// TwinCAT 3 PLC project PLC_ElevatorControl
// ProgramVersion: 3.1.4024.12
// libraries:
//   Tc2_Standard, * (Beckhoff Automation GmbH)
//   Tc2_System, * (Beckhoff Automation GmbH)
//   Tc3_Module, * (Beckhoff Automation GmbH)
//   VisuSymbols,3.5.10.0,System
// project tree:
//   DUTs/ ElevatorOpMode.TcDUT, LiftMovingDirection.TcDUT, txt_opMode.TcTLO
//   / GlobalTextList.TcGTLO, PlcTask.TcTTO, Visualisierungsmanager.TcVMO (not stored)
//   GVLs/ GVL_LiftProj.TcGVL
//   POUs/ FB_ElevatorCtrl.TcPOU, MAIN.TcPOU
//   POUs/POU_ActuatorCtrl/ FB_DriveSimpleDoor.TcPOU, FB_DriveWinch.TcPOU, IF_DriveConstVel.TcIO, IF_DriveVariableVel.TcIO
//   POUs/POU_SequenceCtrl/ FB_move2Level.TcPOU, FB_QM_MinDirChanges.TcPOU, FB_QM_Simple.TcPOU, IF_queueManager.TcIO
//   POUs/POU_Sim/ fb_Aufzug.TcPOU
//   POUs/POU_Util/ FB_BinaryInp.TcPOU, FB_ArrManip.TcPOU
//   VISUs/ Visualization.TcVIS

CONFIGURATION PLC_ElevatorControl
    RESOURCE PLC ON TwinCAT3
        TASK PlcTask(INTERVAL := T#10ms, PRIORITY := 20);
        PROGRAM MAIN WITH PlcTask : MAIN;
    END_RESOURCE
END_CONFIGURATION

// ---- DUTs/ElevatorOpMode.TcDUT
TYPE ElevatorOpMode :
(
	waiting_for_calibration := 0,
	re_init := 1,
	waiting := 2,
	moving := 3,
	doors_opening := 4,
	waiting_doors_open := 5,
	doors_closing := 6,
	prio_waiting := 7,
	prio_doors_closing := 8,
	prio_moving := 9,
	prio_doors_opening := 10
);
END_TYPE

// ---- DUTs/LiftMovingDirection.TcDUT
TYPE LiftMovingDirection :
(
	down := -1,
	up := 1
);
END_TYPE

// ---- GVLs/GVL_LiftProj.TcGVL
VAR_GLOBAL CONSTANT
	NUMLEVELS		:INT	:=4;						(* Total number of levels *)
END_VAR

VAR_GLOBAL
	(* --- User inputs --- *)
	bCallLift 		: ARRAY [1 .. NUMLEVELS] OF BOOL;	(* Assigned to buttons OUTSIDE the lift *)
	bCallLift_Panel : ARRAY [1 .. NUMLEVELS] OF BOOL;	(* Assigned to buttons on the control panel INSIDE the lift *)
	bOpenDoor		: BOOL;
	bCloseDoor		: BOOL;
	
	bSetPrio		: BOOL;								(* For future use *)
	
	(* --- Maintenance variables --- *)
	bInit			: BOOL;
	elOpMode 		: ElevatorOpMode;
END_VAR

// ---- POUs/POU_ActuatorCtrl/IF_DriveConstVel.TcIO
INTERFACE IF_DriveConstVel

METHOD doorClose : BOOL
VAR_INPUT
END_VAR
END_METHOD

METHOD doorDisable
VAR_INPUT
END_VAR
END_METHOD

METHOD doorEnable
VAR_INPUT
END_VAR
END_METHOD

METHOD doorOpen : BOOL
VAR_INPUT
END_VAR
END_METHOD

END_INTERFACE

// ---- POUs/POU_ActuatorCtrl/IF_DriveVariableVel.TcIO
INTERFACE IF_DriveVariableVel

PROPERTY bBOTTOM : BOOL
GET
END_GET
END_PROPERTY

PROPERTY bTOP : BOOL
GET
END_GET
END_PROPERTY

METHOD lifEnable
VAR_INPUT
END_VAR
END_METHOD

METHOD liftDisable
VAR_INPUT
END_VAR
END_METHOD

METHOD moveVarSpeed
VAR_INPUT
	nSetVelocity : INT;
	eDirection : LiftMovingDirection;
END_VAR
END_METHOD

METHOD stop
VAR_INPUT
END_VAR
END_METHOD

END_INTERFACE

// ---- POUs/POU_SequenceCtrl/IF_queueManager.TcIO
INTERFACE IF_queueManager

PROPERTY currentLevel : INT(1..NUMLEVELS)
SET
END_SET
END_PROPERTY

METHOD doneAck
VAR_INPUT
END_VAR
END_METHOD

PROPERTY queue : REFERENCE TO ARRAY [1..NUMLEVELS] OF INT
GET
END_GET
END_PROPERTY

METHOD reset
VAR_INPUT
END_VAR
END_METHOD

END_INTERFACE

// ---- POUs/MAIN.TcPOU
PROGRAM MAIN
VAR
	// actuator control
	smplDoorCtrl		: FB_DriveSimpleDoor;
	winchCtrl 			: FB_DriveWinch;
	
	// simulation
	liftSim				: fb_Aufzug;
	
	// Elevator Controller (main controller)
	// queueLogic			: FB_QM_MinDirChanges;		// sophisticated logic
	queueLogic 			: FB_QM_Simple;				// simple logic
	elevatorCtrl		: FB_ElevatorCtrl;
	
	// processed signals
	bMergedCallBtns 	: ARRAY[1..NUMLEVELS] OF BOOL;

	// utils
	i : INT;
END_VAR

FOR i:=1 TO NUMLEVELS DO
	IF NOT bSetPrio THEN
		bMergedCallBtns[i] := bCallLift[i] OR bCallLift_Panel[i];
	ELSE
		bMergedCallBtns[i] := bCallLift[i];
	END_IF
END_FOR

liftSim(
	bMotorEnable:=winchCtrl.bDriveEnable, 
	nMotorVel:=winchCtrl.nDriveVelocity, 
	bDoorEnable:=smplDoorCtrl.bDriveEnable, 
	bDoorOpen:=smplDoorCtrl.bOpen, 
	bDoorClose:=smplDoorCtrl.bClose, 
	bLiftTop=>winchCtrl.bLimitTop, 
	bLiftBottom=>winchCtrl.bLimitBottom, 
	nLiftPos=> , 
	bDoorIsOpen=>smplDoorCtrl.bLimitSwitchOpen, 
	bDoorIsClosed=>smplDoorCtrl.bLimitSwitchClosed, 
	bLevel0=>elevatorCtrl.bProxSensors[1], 
	bLevel1=>elevatorCtrl.bProxSensors[2], 
	bLevel2=>elevatorCtrl.bProxSensors[3], 
	bLevel3=>elevatorCtrl.bProxSensors[4]);
	
queueLogic(
	bButtons:=bMergedCallBtns
);

elevatorCtrl(
	doorController:=smplDoorCtrl,
	liftController:=winchCtrl,
	queueMngr:=queueLogic,
	bInit_Reinit:=bInit
);

END_PROGRAM

// ---- POUs/POU_ActuatorCtrl/FB_DriveSimpleDoor.TcPOU
FUNCTION_BLOCK FB_DriveSimpleDoor IMPLEMENTS IF_DriveConstVel
VAR_INPUT
	bLimitSwitchOpen, bLimitSwitchClosed : BOOL;		(* Limit switches fpr door open and door closed *)
END_VAR
VAR_OUTPUT
	bDriveEnable, bOpen, bClose : BOOL;					(* Door drive enable, input signals for operning and closing the door *)
END_VAR
VAR
END_VAR

METHOD doorClose : BOOL
(* Close door *)
bClose := TRUE;						(* set outputs for door drive, requires bDoorEnable = TRUE *)
bOpen := FALSE;

doorClose := bLimitSwitchClosed;	(* TRUE if and only if limit switch is TRUE *)
END_METHOD

METHOD doorDisable
bDriveEnable := FALSE;
END_METHOD

METHOD doorEnable
bDriveEnable := TRUE;
END_METHOD

METHOD doorOpen : BOOL
(* Open door *)
bOpen := TRUE;					(* set outputs for door drive, requires bDoorEnable = TRUE *)
bClose := FALSE;

doorOpen := bLimitSwitchOpen;	(* TRUE if and only if limit switch is TRUE *)
END_METHOD

END_FUNCTION_BLOCK

// ---- POUs/POU_ActuatorCtrl/FB_DriveWinch.TcPOU
FUNCTION_BLOCK FB_DriveWinch IMPLEMENTS IF_DriveVariableVel
VAR_INPUT
	bLimitTop, bLimitBottom : BOOL;						(* limit switches *)
END_VAR
VAR_OUTPUT
	bDriveEnable : BOOL;								(* Lift drive enable *)
	nDriveVelocity : INT;								(* Lift drive velocity *)
END_VAR
VAR

END_VAR

PROPERTY bBOTTOM : BOOL
GET
bBOTTOM := bLimitBottom;
END_GET
END_PROPERTY

PROPERTY bTOP : BOOL
GET
bTOP := bLimitTop;
END_GET
END_PROPERTY

METHOD lifEnable
bDriveEnable := TRUE;
END_METHOD

METHOD liftDisable
bDriveEnable := FALSE;
END_METHOD

METHOD moveVarSpeed
VAR_INPUT
	nSetVelocity : INT;						(* velocity setpoint *)
	eDirection : LiftMovingDirection;		(* moving direction: up or down *)
END_VAR
bDriveEnable := TRUE;

IF eDirection > 0 THEN
	eDirection := LiftMovingDirection.up;
END_IF
IF eDirection < 0 THEN
	eDirection := LiftMovingDirection.down; 
END_IF

nSetVelocity := ABS(nSetVelocity);
IF nSetVelocity > 10000 THEN
	nSetVelocity := 10000;
END_IF

IF bLimitTop AND eDirection = LiftMovingDirection.up THEN
	stop();
ELSIF bLimitBottom AND eDirection = LiftMovingDirection.down THEN
	stop();
ELSE
	nDriveVelocity := eDirection*nSetVelocity;
END_IF
END_METHOD

METHOD stop
nDriveVelocity := 0;
END_METHOD

END_FUNCTION_BLOCK

// ---- POUs/POU_Sim/fb_Aufzug.TcPOU
FUNCTION_BLOCK fb_Aufzug
VAR_INPUT
	bMotorEnable 	: BOOL;		(* Deactivate/Activate Motor *)
	nMotorVel 		: INT;
	bDoorEnable 	: BOOL;
	bDoorOpen		: BOOL;
	bDoorClose		: BOOL;
END_VAR
VAR_OUTPUT
	bLiftTop		: BOOL;
	bLiftBottom		: BOOL;
	nLiftPos		: INT(0..1200);
	bDoorIsOpen		: BOOL;
	bDoorIsClosed	: BOOL;
	bLevel0			: BOOL;
	bLevel1			: BOOL;
	bLevel2			: BOOL;
	bLevel3			: BOOL;
END_VAR
VAR
	nMotorSpeed		: INT;
	nDoorPos		: INT(0..100);
	bInit			: BOOL := FALSE;
	tDoorsClosing	: TIME := T#180MS;
	tDoorsOpening	: TIME := T#220MS;
	tS2T			: TIME;
	tDoorDelay		: TON;
	tMovingDelay	: TON;
END_VAR

(* Initial sensor outputs *)
IF NOT bInit THEN
	bInit := TRUE;
	bLevel0 := TRUE;
	bLevel1 := FALSE;
	bLevel2 := FALSE;
	bLevel3 := FALSE;
	nLiftPos := 0;
	nDoorPos := 100;		(* 100 means door open, 0 is closed *)
	bLiftBottom := TRUE;
	bLiftTop := FALSE;
	bDoorIsOpen := TRUE;
	bDoorIsClosed := FALSE;
END_IF

(* Limiting Motor speed *)
IF nMotorVel > 10000 THEN
	nMotorVel := 10000;
ELSIF nMotorVel < -10000 THEN
	nMotorVel := -10000;
END_IF
nMotorSpeed := ABS(nMotorVel);

(* Lift behavior *)
IF nLiftPos = 1200 THEN
	bLiftTop := TRUE;
	bLevel3 := TRUE;
ELSIF nLiftPos = 0 THEN
	bLiftBottom := TRUE;
	bLevel0 := TRUE;
ELSE
	bLiftTop := FALSE;
	bLiftBottom := FALSE;
END_IF

IF NOT bMotorEnable THEN
	(* Remain position and do noting *)
ELSE
	(* Calculate delay, after which the pos should be increased by 10.
	 Note that delay should be lager the lower nMotorSpeed is.
	 The calculations here yield a total duration from 0 to maxPos of 
	approx. 4.8 seconds with 10000 nMotorVel *)
	IF nMotorSpeed <> 0 THEN
		tS2T := INT_TO_TIME((12000-nMotorSpeed)/50);
		tMovingDelay(IN:=TRUE, PT:=tS2T);
		IF tMovingDelay.Q THEN
			tMovingDelay(IN:=FALSE);
			IF nMotorVel > 0 AND nLiftPos < 1200 THEN
				nLiftPos := nLiftPos + 10; 
			ELSIF nMotorVel < 0 AND nLiftPos > 0 THEN
				nLiftPos := nLiftPos - 10;
			END_IF
			
			IF nLiftPos = 0 OR nLiftPos = 60 THEN
				bLevel0 := TRUE;
			ELSIF nLiftPos = 340 OR nLiftPos = 400 OR nLiftPos = 460 THEN
				bLevel1 := TRUE;
			ELSIF nLiftPos = 740 OR nLiftPos = 800 OR nLiftPos = 860 THEN
				bLevel2 := TRUE;
			ELSIF nLiftPos = 1140 OR nLiftPos = 1200 THEN
				bLevel3 := TRUE;
			ELSE
				bLevel0 := FALSE;
				bLevel1 := FALSE;
				bLevel2 := FALSE;
				bLevel3 := FALSE;
			END_IF
		END_IF
	END_IF
END_IF


(* Door dynamics *)
IF bDoorEnable THEN
	IF bDoorOpen AND NOT bDoorClose AND nDoorPos < 100 THEN
		tDoorDelay(IN:=TRUE, PT:=tDoorsOpening);
		IF tDoorDelay.Q THEN
			tDoorDelay(IN:=FALSE);
			nDoorPos := nDoorPos + 10;
		END_IF
	ELSIF bDoorClose AND NOT bDoorOpen AND nDoorPos > 0 THEN
		tDoorDelay(IN:=TRUE, PT:=tDoorsClosing);
		IF tDoorDelay.Q THEN
			tDoorDelay(IN:=FALSE);
			nDoorPos := nDoorPos - 10;
		END_IF
	END_IF
END_IF

(* set door state *)
IF nDoorPos = 100 THEN
	bDoorIsOpen := TRUE;
ELSIF nDoorPos = 0 THEN
	bDoorIsClosed := TRUE;
ELSE
	bDoorIsOpen := FALSE;
	bDoorIsClosed := FALSE;
END_IF

END_FUNCTION_BLOCK

// ---- POUs/POU_SequenceCtrl/FB_QM_Simple.TcPOU
FUNCTION_BLOCK FB_QM_Simple IMPLEMENTS IF_queueManager
VAR_INPUT
	bButtons 	  : ARRAY [1..NUMLEVELS] OF BOOL;						(* user input *)
END_VAR
VAR_OUTPUT
END_VAR
VAR
	tPushDetects  : ARRAY [1..NUMLEVELS] OF FB_BinaryInp;				(* FBs to buffer user inputs until being processed *)
	queueManip	  : FB_ArrManip;										(* FB for array manipulation, like sorting etc. *)
	k			  : INT;												(* loop variable *)
	
	nCurLevel	  : INT(1..NUMLEVELS);									(* current lift position *)
	nQueue		  : ARRAY [1..NUMLEVELS] OF INT;						(* queue, saving next targets in current moving direction *)
	bLevelInQueue : ARRAY [1..NUMLEVELS] OF BOOL;						(* buffer of all active calls , i.e. levels in nQueue OR active tPushDetects *)
END_VAR

FOR k:=1 TO NUMLEVELS DO
	tPushDetects[k](bPush:=bButtons[k], bReset:=FALSE);
	bLevelInQueue[k] := tPushDetects[k].bOutActive OR queueManip.isElement(arr:=nQueue, entry:=k);
END_FOR

FOR k:=1 TO NUMLEVELS DO
	IF tPushDetects[k].bOutActive THEN
		IF NOT queueManip.isElement(arr:=nQueue, entry:=k) THEN
			// Inset new element
			queueManip.insert(arr:=nQueue, newElement:=k, freeElement:=0);
		END_IF	
	
		// Then acknowledge
		tPushDetects[k](bReset:=TRUE);
	END_IF
END_FOR

PROPERTY currentLevel : INT (1..NUMLEVELS)
SET
nCurLevel := currentLevel;
END_SET
END_PROPERTY

METHOD doneAck
VAR_INPUT
END_VAR
VAR
END_VAR
(* 
By calling this method, the first entry in nQueue is deleted and all remaining entries are shiftetd one position forward. 
Method shall be called, after the latest moving job has been executed. 
*)
queueManip.pop_front(arr:=nQueue, fill:=0);
END_METHOD

PROPERTY queue : REFERENCE TO ARRAY [1..NUMLEVELS] OF INT
GET
queue REF= nQueue;
END_GET
END_PROPERTY

METHOD reset
VAR_INPUT
END_VAR
VAR
	i : INT;
END_VAR
(* resets all calls *)
FOR i:=1 TO NUMLEVELS DO
	nQueue[i] := 0;
	tPushDetects[i](bReset:=TRUE);
END_FOR
END_METHOD

END_FUNCTION_BLOCK

// ---- POUs/POU_Util/FB_BinaryInp.TcPOU
FUNCTION_BLOCK FB_BinaryInp
VAR_INPUT
	bPush : BOOL;
	bReset : BOOL;
END_VAR
VAR_OUTPUT
	bOutActive : BOOL;
END_VAR
VAR
	rsHold : RS;
END_VAR

rsHold(SET:=bPush, RESET1:=bReset, Q1=>bOutActive);

END_FUNCTION_BLOCK

// ---- POUs/POU_Util/FB_ArrManip.TcPOU
FUNCTION_BLOCK FB_ArrManip
VAR_INPUT
END_VAR
VAR_OUTPUT
END_VAR
VAR
END_VAR

METHOD flip
VAR_INPUT
	arr : REFERENCE TO ARRAY [1..NUMLEVELS] OF INT;
END_VAR
VAR
	i, mid : INT;
	bfr : INT;
END_VAR
mid := NUMLEVELS/2;
FOR i:=1 TO mid DO
	bfr := arr[i];
	arr[i] := arr[NUMLEVELS+1-i];
	arr[NUMLEVELS+1-i] := bfr;
END_FOR
END_METHOD

METHOD index : INT
VAR_INPUT
	arr : REFERENCE TO ARRAY [1..NUMLEVELS] OF BOOL;
END_VAR
VAR
	i : INT;
END_VAR
(* 
Method returns the index of the first element that is TRUE.
If all Elements are zero, the return value is 0.
*)

FOR i:=1 TO NUMLEVELS DO
	IF arr[i] = TRUE THEN
		index := i;
		RETURN;
	END_IF
END_FOR

index := 0;
END_METHOD

METHOD insert : BOOL
VAR_INPUT
	arr : REFERENCE TO ARRAY [1..NUMLEVELS] OF INT;
	newElement : INT;
	freeElement : INT;
END_VAR
VAR 
	i : INT;
END_VAR
FOR i:=1 TO NUMLEVELS DO
	IF arr[i] = newElement THEN
		insert := TRUE;
		RETURN;
	END_IF
END_FOR

FOR i:=1 TO NUMLEVELS DO
	IF arr[i] = freeElement THEN
		arr[i] := newElement;
		insert := TRUE;
		RETURN;
	END_IF
END_FOR

insert := FALSE;
END_METHOD

METHOD isElement : BOOL
VAR_INPUT
	arr : REFERENCE TO ARRAY [1..NUMLEVELS] OF INT;
	entry : INT;
END_VAR
VAR
	i : INT;
END_VAR
FOR i:=1 TO NUMLEVELS DO
	IF arr[i] = entry THEN
		isELement := TRUE;
		RETURN;
	END_IF
END_FOR
isElement := FALSE;
END_METHOD

METHOD isEmpty : BOOL
VAR_INPUT
	arr : REFERENCE TO ARRAY [1..NUMLEVELS] OF INT;
	emptyElement : INT;
END_VAR
VAR
	i : INT;
END_VAR
FOR i:=1 TO NUMLEVELS DO
	IF arr[i] <> emptyElement THEN
		isEmpty := FALSE;
		RETURN;
	END_IF
END_FOR
isEmpty := TRUE;
END_METHOD

METHOD PRIVATE partition : INT
VAR_INPUT
	arr : REFERENCE TO ARRAY [1..NUMLEVELS] OF INT;
	lo, hi : INT;
END_VAR
VAR
	pivot : INT;
	i, j : INT;
	bfr : INT;
END_VAR
pivot := arr[hi];
i := lo;

FOR j:=lo TO hi DO
	IF arr[j] < pivot THEN
		bfr := arr[i];
		arr[i] := arr[j];
		arr[j] := bfr;
		i := i+1;
	END_IF
END_FOR

bfr := arr[i];
arr[i] := arr[hi];
arr[hi] := bfr;

partition := i;
END_METHOD

METHOD pop_front : INT
VAR_INPUT
	arr : REFERENCE TO ARRAY [1..NUMLEVELS] OF INT;
	fill : INT;
END_VAR
VAR
	nOut : INT;
	i : INT;
END_VAR
nOut := arr[1];

FOR i:=1 TO NUMLEVELS-1 DO
	arr[i] := arr[i+1];
END_FOR
arr[NUMLEVELS] := fill;

pop_front := nOut;
END_METHOD

METHOD quicksort_asc
VAR_INPUT
	arr : REFERENCE TO ARRAY [1..NUMLEVELS] OF INT;
	lo, hi : INT;
END_VAR
VAR
	p : INT;
END_VAR
IF lo < hi THEN
	p := partition(arr, lo, hi);
	quicksort_asc(arr, lo, p-1);
	quicksort_asc(arr, p+1, hi);
END_IF
END_METHOD

METHOD quicksort_desc
VAR_INPUT
	arr : REFERENCE TO ARRAY [1..NUMLEVELS] OF INT;
	lo, hi : INT;
END_VAR
VAR
	p : INT;
END_VAR
quicksort_asc(arr:=arr, lo:=lo, hi:=hi);
flip(arr:=arr);
END_METHOD

END_FUNCTION_BLOCK

// ---- POUs/FB_ElevatorCtrl.TcPOU
(* 
	FB_ElevatorCtrl is the main control unit which orchestrates the process steps
*)
FUNCTION_BLOCK FB_ElevatorCtrl
VAR_INPUT
	// controlling actuators 
	doorController 		: IF_DriveConstVel;
	liftController 		: IF_DriveVariableVel;
	
	// functionalities
	queueMngr			: IF_queueManager;				// orchestrates btn calls and manages which level is appraoched next
	
	// maintenance
	bInit_Reinit 		: BOOL;
	
	// system outputs (from simulation FB)
	bProxSensors		: ARRAY [1..NUMLEVELS] OF BOOL;
	
END_VAR
VAR_OUTPUT
	// for maintenance and VISU
	operationMode 		: ElevatorOpMode;
	bError				: BOOL;
END_VAR
VAR
	levelController 	: FB_move2Level;				// moves lift to next position
	arrUtil				: FB_ArrManip;					// array manipulation (used in ln. 3 only)
	nState 				: INT;							// state no. of state diagram
	
	// Timer
	tWait				: TON;							// waiting time, used in calibration mode (init)
	tDoorOpen			: TON;
	
	// trigger detections
	trInitDetect 		: R_TRIG;
	trJobDone			: R_TRIG;
	trOpenDoor			: R_TRIG;
	
	// local bfr variables
	curLevel 			: INT(1..NUMLEVELS);
	locBfrQueue			: ARRAY [1..NUMLEVELS] OF INT;
	bBfrDoorState		: BOOL;

	// next level in prio mode
	prioNextLevel		: INT(0..NUMLEVELS) := 0;
	prioArrManip 		: FB_ArrManip;
END_VAR

trInitDetect(CLK:=bInit_Reinit);									// trigger for calling maintenance state (active in idle mode only)
trOpenDoor(CLK:=bOpenDoor);											// trigger for push btn: OPEN DOOR
IF arrUtil.index(arr:=bProxSensors) <> 0 THEN
	curLevel := arrUtil.index(arr:=bProxSensors);					// detetct current lift position -> translate binary signal of prox sensor to int
END_IF
queueMngr.currentLevel := curLevel;									// passing current level to Queue Manager


CASE nState OF
	0:		// idle
		operationMode := ElevatorOpMode.waiting_for_calibration;
		IF trInitDetect.Q THEN
			operationMode := ElevatorOpMode.re_init;
			nState := 101;											// maintenance mode
		END_IF
		
	1:		// nominal operation mode: waiting
		operationMode := ElevatorOpMode.waiting;
		locBfrQueue := queueMngr.queue;								// update queue		
		IF bSetPrio THEN
			nState := 21;											// switch to prio mode
		ELSE
			IF locBfrQueue[1] <> 0 THEN								// queue is not empty -> start moving
				levelController(bStart:=FALSE);
				nState := 2;
			END_IF
			IF trOpenDoor.Q THEN
				nState := 13;										// push btn DOOR OPEN possible only when lift is in waiting mode
			END_IF
		END_IF				
		
		IF trInitDetect.Q THEN
			operationMode := ElevatorOpMode.re_init;
			nState := 101;											// maintenance mode
		END_IF
		
		
	2:		// nominal operation mode: move to next level
		operationMode := ElevatorOpMode.moving;
		locBfrQueue := queueMngr.queue;								// update queue: New calls, which pop up while lift is already moving, are considered
		levelController(
			winchCtrl:=liftController,
			bProxSensor:=bProxSensors,
			bStart:=TRUE,
			nCurrentLevel:=curLevel,
			nNextLevel:=locBfrQueue[1]
			);														// calling FB starts moving until job is done
		trJobDone(CLK:=levelController.bJobDone);					// trigger for detection "job done"-signal
		
		IF trJobDone.Q THEN
			levelController(bStart:=FALSE);							// set bStart to FALSE is necessary to start new job
			doorController.doorEnable();							
			nState := 3;
		END_IF
		
		(*
			POSSIBLE IMPROVEMENT:
			Steps 3 - 5 (as well as 13 - 15) are used for controlling to lift doors. It would be better to
			outsource this process control steps to a separate FB, similarly to FB_move2Level. That would 
			open up the possibilty for using different "door moving logics", like a new door with a light barrier.
		*)
		
	3:		// nominal operation mode: open door at target level
		operationMode := ElevatorOpMode.doors_opening;
		bBfrDoorState := doorController.doorOpen();
		IF bBfrDoorState THEN
			nState:=4;
		END_IF
			
	4:		// nominal operation mode: keep door open for 3sec
		operationMode := ElevatorOpMode.waiting_doors_open;
		tDoorOpen(IN:=TRUE, PT:=T#3S);								// duration fordoor being open is fixed (3sec)
		IF tDoorOpen.Q THEN
			tDoorOpen(IN:=FALSE);
			nState := 5;
		END_IF
		
	5:		// nominal operation mode: close doors
		operationMode := ElevatorOpMode.doors_closing;
		bBfrDoorState := doorController.doorClose();
		IF bBfrDoorState THEN
			doorController.doorDisable();
			IF bSetPrio THEN
				nState := 21;
				prioNextLevel := 0;
			ELSE
				queueMngr.doneAck();
				nState := 1;
			END_IF
		END_IF	
	
	13:		// nominal operation mode: open door at target level
		operationMode := ElevatorOpMode.doors_opening;
		doorController.doorEnable();
		bBfrDoorState := doorController.doorOpen();
		IF bBfrDoorState THEN
			nState:=14;
		END_IF
			
	14:		// nominal operation mode: keep door open for 3sec
		operationMode := ElevatorOpMode.waiting_doors_open;
		tDoorOpen(IN:=TRUE, PT:=T#3S);
		IF tDoorOpen.Q THEN
			tDoorOpen(IN:=FALSE);
			nState := 15;
		END_IF
		
	15:		// nominal operation mode: close doors
		operationMode := ElevatorOpMode.doors_closing;
		bBfrDoorState := doorController.doorClose();
		IF bBfrDoorState THEN
			doorController.doorDisable();
			nState := 1;
		END_IF	
		
	21:		// PRIO mode: waiting for call
		operationMode := ElevatorOpMode.prio_waiting;
		prioNextLevel := 0;
		IF NOT bSetPrio THEN
			nState := 1;											// switch to normal mode
		ELSE
			prioNextLevel := prioArrManip.index(arr:=bCallLift_Panel);
			IF prioNextLevel <> 0 THEN
				nState := 22;
			END_IF
		END_IF

	22:		// PRIO mode: close doors
		operationMode := ElevatorOpMode.prio_doors_closing;
		bBfrDoorState := doorController.doorClose();
		IF bBfrDoorState THEN
			doorController.doorDisable();
			nState := 23;
		END_IF	
		
	23:		// PRIO mode: moving
		operationMode := ElevatorOpMode.prio_moving;
		levelController(
			winchCtrl:=liftController,
			bProxSensor:=bProxSensors,
			bStart:=TRUE,
			nCurrentLevel:=curLevel,
			nNextLevel:=prioNextLevel
			);														// calling FB starts moving until job is done
		trJobDone(CLK:=levelController.bJobDone);					// trigger for detection "job done"-signal
		
		IF trJobDone.Q THEN
			levelController(bStart:=FALSE);							// set bStart to FALSE is necessary to start new job
			doorController.doorEnable();							
			nState := 3;
		END_IF
		
	101:	// re_init: stop elevator and clear queue callStates
		queueMngr.reset();
		liftController.stop();
		doorController.doorEnable();
		IF doorController.doorClose() THEN
			nState := 102;
		END_IF
		
	102:	// stop for a few seconds, then move down
		tWait(IN:=TRUE, PT:=T#2S);
		IF tWait.Q THEN
			nState := 103;
		END_IF

	103:	// re_init: Move elevator to bottom
		liftController.moveVarSpeed(nSetVelocity:=5000, eDirection:=LiftMovingDirection.down);		(* Move down fast *);
		IF liftController.bBOTTOM THEN
			// controller stops lift (cf. method moveVarSpeed)
			// curLevel should now be 1
			IF curLevel <> 1 THEN
				bError := TRUE;
			ELSE
				bError := FALSE;
			END_IF
			nState := 1;			// go to normal operation mode
		END_IF
		
		
END_CASE

END_FUNCTION_BLOCK

// ---- POUs/POU_SequenceCtrl/FB_move2Level.TcPOU
FUNCTION_BLOCK FB_move2Level
VAR_INPUT
	winchCtrl : REFERENCE TO IF_DriveVariableVel;		(* function block for controlling winch drive *)
	bProxSensor : ARRAY [1..NUMLEVELS] OF BOOL;			(* Proximity sensors for level L0 .. L_NUMLEVELS *)
	bStart : BOOL;										(* Signal to start moving *)
	
	nCurrentLevel : INT(1..NUMLEVELS);					(* current lift position *)
	nNextLevel : INT(1..NUMLEVELS);						(* setpoint of next target -> first entry of queue *)
END_VAR
VAR_OUTPUT
	bJobDone : BOOL := FALSE;							(* feedback when target is reached: signal is TRUE for one cycle *)
END_VAR
VAR
	eDirection : LiftMovingDirection;					(* local variable for lift moving direction *)
	
	nState : INT := 0;									(* state variable for sequential control *)
	nCnt : INT;											(* loop variable *)
	
	tLevelDetection : R_TRIG;							(* trigger used fpr proximity sensors *)
	tStartDetection : R_TRIG;							(* trigger for detecting start signal *)
END_VAR
VAR CONSTANT
	nVelFast : INT := 5000;								(* setpoints for fast and slow moving *)
	nVelSlow : INT := 10;
END_VAR

tStartDetection(CLK:=bStart);

CASE nState OF
	0:	// idle -> lift is waiting for start signal
		bJobDone := FALSE;
		IF tStartDetection.Q THEN
			nState := 1;								(* start next job *)
		END_IF
		
	1: 	// set direction
		bJobDone := FALSE;
		IF nNextLevel < nCurrentLevel THEN				(* move down to get to next level *)
			eDirection := LiftMovingDirection.down;
			nState := 2;
		END_IF
		IF nNextLevel > nCurrentLevel THEN				(* move up to get to next level *)
			eDirection := LiftMovingDirection.up;
			nState := 2;
		END_IF
		IF nNextLevel = nCurrentLevel THEN				(* lift is already in right position *)
			bJobDone := TRUE;
			nState := 0;
		END_IF
		
	2:	// move up/down slowly - START
		winchCtrl.moveVarSpeed(nSetVelocity:=nVelSlow, eDirection:=eDirection);
		tLevelDetection(CLK:=bProxSensor[nCurrentLevel]);
		IF tLevelDetection.Q THEN
			nState := 3;
		END_IF
		
	3: 	// move up/down fast
		winchCtrl.moveVarSpeed(nSetVelocity:=nVelFast, eDirection:=eDirection);
		tLevelDetection(CLK:=bProxSensor[nNextLevel]);
		IF tLevelDetection.Q THEN
			nState := 4;
		END_IF
		
	4:	// move up/down slowly - END
		winchCtrl.moveVarSpeed(nSetVelocity:=nVelSlow, eDirection:=eDirection);
		tLevelDetection(CLK:=bProxSensor[nNextLevel]);
		IF tLevelDetection.Q THEN
			winchCtrl.stop();
			bJobDOne := TRUE;
			nState := 0;									(* moving job completed: go back to idle state *)
		END_IF
		
END_CASE

END_FUNCTION_BLOCK

// ---- POUs/POU_SequenceCtrl/FB_QM_MinDirChanges.TcPOU
FUNCTION_BLOCK FB_QM_MinDirChanges IMPLEMENTS IF_queueManager
VAR_INPUT
	bButtons 	  : ARRAY [1..NUMLEVELS] OF BOOL;						(* user input *)
END_VAR
VAR_OUTPUT
END_VAR
VAR
	tPushDetects  : ARRAY [1..NUMLEVELS] OF FB_BinaryInp;				(* FBs to buffer user inputs until being processed *)
	queueManip	  : FB_ArrManip;										(* FB for array manipulation, like sorting etc. *)
	k			  : INT;												(* loop variable *)
	eDirection    : LiftMovingDirection := LiftMovingDirection.up;		(* local variable for moving direction *)
	
	nCurLevel	  : INT(1..NUMLEVELS);									(* current lift position *)
	nQueue		  : ARRAY [1..NUMLEVELS] OF INT;						(* queue, saving next targets in current moving direction *)
	bLevelInQueue : ARRAY [1..NUMLEVELS] OF BOOL;						(* buffer of all active calls , i.e. levels in nQueue OR active tPushDetects *)
END_VAR

FOR k:=1 TO NUMLEVELS DO
	tPushDetects[k](bPush:=bButtons[k], bReset:=FALSE);
	bLevelInQueue[k] := tPushDetects[k].bOutActive OR queueManip.isElement(arr:=nQueue, entry:=k);
END_FOR

FOR k:=1 TO NUMLEVELS DO
	IF tPushDetects[k].bOutActive THEN
		IF queueManip.isEmpty(arr:=nQueue, emptyElement:=0) THEN
			// Queue is empty. Just inset new element and sort desc (-> new Element is at front)
			queueManip.insert(arr:=nQueue, newElement:=k, freeElement:=0);
			queueManip.quicksort_desc(arr:=nQueue, lo:=1, hi:=NUMLEVELS);
			// ... and set Direction to UP if current lift position is below the calling level
			IF nCurLevel < k THEN
				eDirection := LiftMovingDirection.up;
			END_IF
			// ... and set Direction to DOWN if current lift position is above the calling level
			IF nCurLevel > k THEN
				eDirection := LiftMovingDirection.down;
			END_IF
			// otherwise leave direction as it is!
			
			// Then acknowledge
			tPushDetects[k](bReset:=TRUE);
			CONTINUE;
		END_IF	
	
		(*
			if new call is already included in queue, then acknowldge
			and continue with next loop iteration 
		*)
		IF queueManip.isElement(arr:=nQueue, entry:=k) THEN
			tPushDetects[k](bReset:=TRUE);
			CONTINUE;
		END_IF
		
		(* 
			lift is moving up and new call is from above the lift position,
			so the new call in inserted into queue and queue is sorted afterwards.
		*)
		IF nCurLevel < k AND eDirection = LiftMovingDirection.up THEN
			queueManip.insert(arr:=nQueue, newElement:=k, freeElement:=0);
			queueManip.quicksort_asc(arr:=nQueue, lo:=1, hi:=NUMLEVELS);
			WHILE nQueue[1] = 0 DO
				queueManip.pop_front(arr:=nQueue, fill:=0);
			END_WHILE
			// ack call
			tPushDetects[k](bReset:=TRUE);
		END_IF
		
		(* 
			lift is moving down and new call is from below the lift position,
			so the new call in inserted into queue and queue is sorted afterwards.
		*)
		IF nCurLevel > k AND eDirection = LiftMovingDirection.down THEN
			queueManip.insert(arr:=nQueue, newElement:=k, freeElement:=0);
			queueManip.quicksort_desc(arr:=nQueue, lo:=1, hi:=NUMLEVELS);
			// ack call
			tPushDetects[k](bReset:=TRUE);
		END_IF
	END_IF
END_FOR

PROPERTY currentLevel : INT (1..NUMLEVELS)
SET
nCurLevel := currentLevel;
END_SET
END_PROPERTY

METHOD doneAck
VAR_INPUT
END_VAR
VAR
END_VAR
(* 
By calling this method, the first entry in nQueue is deleted and all remaining entries are shiftetd one position forward. 
Method shall be called, after the latest moving job has been executed. 
*)
queueManip.pop_front(arr:=nQueue, fill:=0);
END_METHOD

PROPERTY queue : REFERENCE TO ARRAY [1..NUMLEVELS] OF INT
GET
queue REF= nQueue;
END_GET
END_PROPERTY

METHOD reset
VAR_INPUT
END_VAR
VAR
	i : INT;
END_VAR
(* resets all calls *)
FOR i:=1 TO NUMLEVELS DO
	nQueue[i] := 0;
	tPushDetects[i](bReset:=TRUE);
END_FOR
END_METHOD

END_FUNCTION_BLOCK

// ---- DUTs/txt_opMode.TcTLO
TEXTLIST txt_opMode
  0 = 'waiting_for_calibration'
  1 = 're_init'
  2 = 'waiting'
  3 = 'moving'
  4 = 'doors_opening'
  5 = 'waiting_doors_open'
  6 = 'doors_closing'
  7 = 'PRIO waiting'
  8 = 'PRIO doors_closing'
  9 = 'PRIO moving'
  10 = 'PRIO doors_opening'
   = ''
END_TEXTLIST

// ---- GlobalTextList.TcGTLO
TEXTLIST GlobalTextList
  97 = 'Bedienpanel'
  895 = 'Calibrate'
  874 = 'Ebene 0'
  118 = 'Ebene 1'
  419 = 'Ebene 2'
  935 = 'Ebene 3'
  213 = 'Ebene 4'
  843 = 'Erdgeschoss'
  728 = 'Maintenance'
  676 = 'Moving direction:'
  634 = 'Operation state:'
  75 = 'PRIO'
  113 = 'PRIOauf'
  853 = 'Queue:'
  392 = 'Start Calibrate'
  811 = 'Start calibration'
  225 = 'Start calibration:'
  373 = 'Tür auf'
  901 = 'Tür auf0'
END_TEXTLIST

// ---- VISUs/Visualization.TcVIS
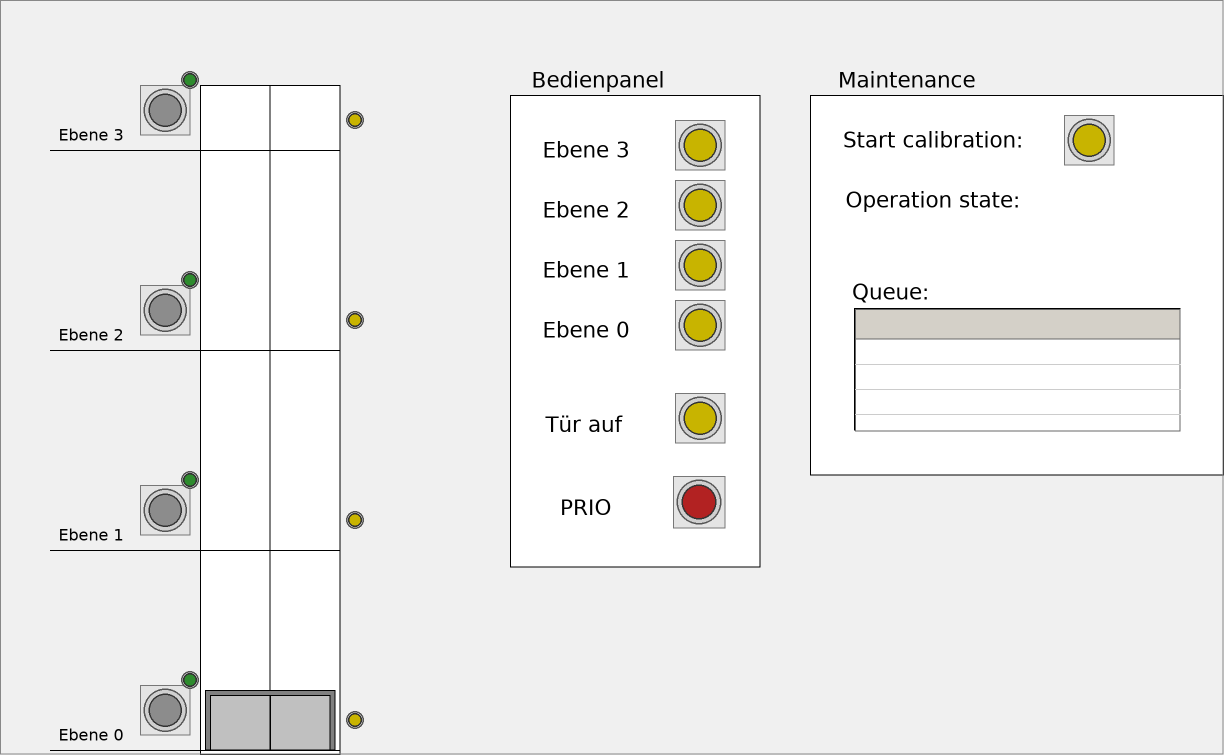
VISUALIZATION Visualization  // 1224x755
    RoundedRectangle (510,95 250x472)
    Lamp1 (345,710 20x20), variable: MAIN.elevatorCtrl.bProxSensors[1], style: Lamp-Lamp1-Yellow
    Rectangle (200,85 140x670)
    Lamp1 (345,510 20x20), variable: MAIN.elevatorCtrl.bProxSensors[2], style: Lamp-Lamp1-Yellow
    Lamp1 (345,310 20x20), variable: MAIN.elevatorCtrl.bProxSensors[3], style: Lamp-Lamp1-Yellow
    Lamp1 (345,110 20x20), variable: MAIN.elevatorCtrl.bProxSensors[4], style: Lamp-Lamp1-Yellow
    Line (50,750) (340,750)
    Line (50,550) (340,550)
    Line (50,350) (340,350)
    Line (50,150) (340,150)
    Label (50,120 82x30), "Ebene 3"
    Label (50,320 82x30), "Ebene 2"
    Label (50,520 82x30), "Ebene 1"
    Label (50,720 82x30), "Ebene 0"
    Rectangle (205,690 130x60)
        p2738717112: -MAIN.liftSim.nLiftPos/2
    Rectangle (210,695 120x55)
        p2738717112: -MAIN.liftSim.nLiftPos/2
    Rectangle (210,695 60x55)
        p874137650: -MAIN.liftSim.nDoorPos/2
        p2738717112: -MAIN.liftSim.nLiftPos/2
    Rectangle (270,695 60x55)
        p2738717112: -MAIN.liftSim.nLiftPos/2
        p3528305787: MAIN.liftSim.nDoorPos/2
    PushSwitch (140,285 50x50), variable: bCallLift[3], behaviour: TAP, style: Switch-PushSwitch-Gray
    PushSwitch (140,85 50x50), variable: bCallLift[4], behaviour: TAP, style: Switch-PushSwitch-Gray
    PushSwitch (140,485 50x50), variable: bCallLift[2], behaviour: TAP, style: Switch-PushSwitch-Gray
    PushSwitch (140,685 50x50), variable: bCallLift[1], behaviour: TAP, style: Switch-PushSwitch-Gray
    PushSwitch (675,120 50x50), variable: bCallLift_Panel[4], behaviour: TAP, style: Switch-PushSwitch-Yellow
    Label (545,135 82x30), "Ebene 3"
    Label (545,195 82x30), "Ebene 2"
    PushSwitch (675,180 50x50), variable: bCallLift_Panel[3], behaviour: TAP, style: Switch-PushSwitch-Yellow
    PushSwitch (675,240 50x50), variable: bCallLift_Panel[2], behaviour: TAP, style: Switch-PushSwitch-Yellow
    Label (545,255 82x30), "Ebene 1"
    Label (545,315 82x30), "Ebene 0"
    PushSwitch (675,300 50x50), variable: bCallLift_Panel[1], behaviour: TAP, style: Switch-PushSwitch-Yellow
    Label (541,408 86x33), "Tür auf"
    Label (498,65 200x30), "Bedienpanel"
    RoundedRectangle (810,95 414x380)
    Label (807,65 200x30), "Maintenance"
    Label (850,125 166x30), "Start calibration:"
    PushSwitch (1064,115 50x50), variable: bInit, behaviour: TAP, style: Switch-PushSwitch-Yellow
    Label (843,185 180x30), "Operation state:"
    Label (843,220 347x40)
    Rectangle (845,219 354x30), text list: 'txt_opMode', text index: MAIN.elevatorCtrl.operationMode
    PushSwitch (675,393 50x50), variable: bOpenDoor, behaviour: TAP, style: Switch-PushSwitch-Yellow
    Rectangle (854,308 326x122)
    Table (855,309 325x122), data array: MAIN.queueLogic.nQueue
        p3854506369: MAIN.queueLogic.nQueue[INDEX]
    Label (843,277 95x30), "Queue:"
    Lamp1 (180,670 20x20), variable: MAIN.queueLogic.bLevelInQueue[1], style: Lamp-Lamp1-Green
    Lamp1 (180,470 20x20), variable: MAIN.queueLogic.bLevelInQueue[2], style: Lamp-Lamp1-Green
    Lamp1 (180,270 20x20), variable: MAIN.queueLogic.bLevelInQueue[3], style: Lamp-Lamp1-Green
    Lamp1 (180,70 20x20), variable: MAIN.queueLogic.bLevelInQueue[4], style: Lamp-Lamp1-Green
    Line (270,690) (270,85)
        p2773130477: -MAIN.liftSim.nLiftPos/2
    Label (543,491 86x33), "PRIO"
    PushSwitch (673,476 52x52), variable: bSetPrio, behaviour: TOGGLE, style: Switch-PushSwitch-Red
END_VISUALIZATION
